Fanuc KAREL source: ko00051.KL

PROGRAM KO00051
%STACKSIZE=65535
%PRIORITY=65535
%NOLOCKGROUP
VAR
P1 : XYZWPR
P2 : POSITION
F : BOOLEAN
OUT : XYZWPREXT
BEGIN
F=TRUE
-- UNSAFE_SOURCE_IR line 11: OUT = MIRROR(convert_xyzwpr_to_xyzwprext(P1), P2, F)
END KO00051
